TYPE ST_AxisSpg :
STRUCT
    AXIS : AXIS_REF;
    spgEnable : MC_ExtSetPointGenEnable;
    spgDisable : MC_ExtSetPointGenDisable;
    position : LREAL;
    velocity : LREAL;
    direction : DINT;
END_STRUCT
END_TYPE

(* stored: Version 1.1.0.1, ProductVersion 3.1.4024.11
   DUT ST_AxisSpg: Id {305aec02-ecf2-465e-96a1-4235bd4322b7} *)
